Fanuc KAREL source: kd00067.KL

-- PROVISIONAL review KL for V1013-1; original PC SHA256 028217ff09e9f3ebdec573f2f5243070206113cc0566bad83643dd3f846e5e78
-- Incomplete behavior may be omitted. Consult companion uncertainty JSON. Do not deploy.
PROGRAM KD00067
%NOLOCKGROUP
VAR
  I : INTEGER
  J : INTEGER
  B : BOOLEAN
  R : REAL
  S : STRING[80]
BEGIN
  -- UNRESOLVED_PC offsets 5-18; opcodes 9D,81,18,9D,1B,9D,12,9C,13,04
  -- UNRESOLVED_PC offsets 23-27; opcodes 7F
END KD00067
